RoboDK station: MoveBill_V2.rdk

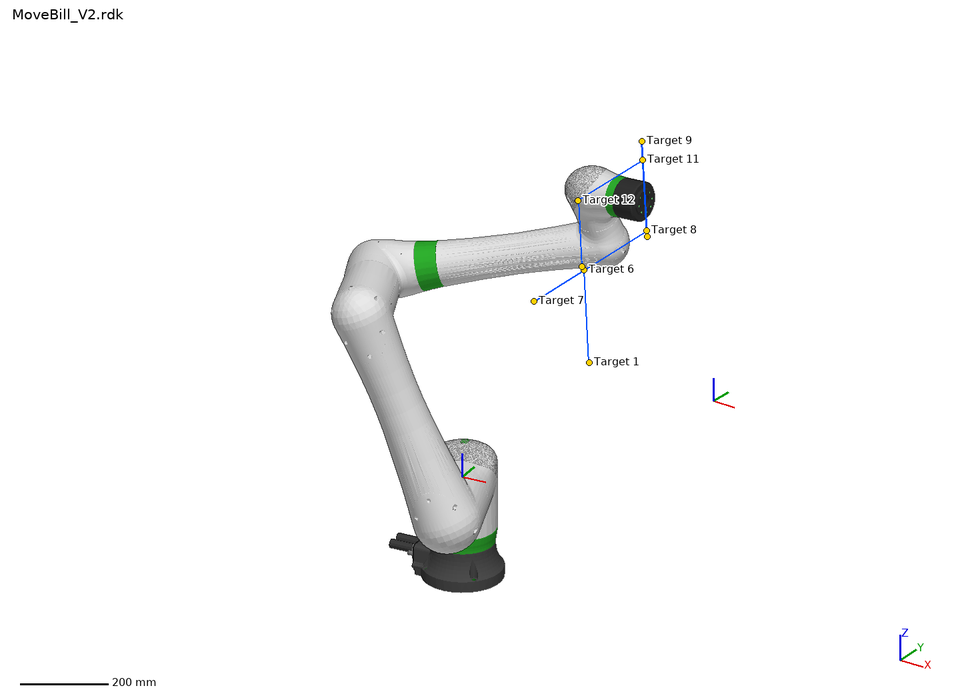
[picture v0: the station drawn from its stored meshes, robots at their saved joint values, targets as dots, program paths as lines]
Station MoveBill_V2 (saved by RoboDK 5.5.4). Poses are relative to the parent item; angles as X-Y-Z fixed-axis rotations.
Station parameters (name, value as stored): LIN64
  - frame Fanuc CRX-10iA Base at (0, 0, 245) mm, rotated rx 0 ry 0 rz 7.43 deg
    - robot Fanuc CRX-10iA: 6 axes, payload 10 kg, reach 1249 mm, repeatability 0.05 mm, weight 40 kg
        modified DH rows (alpha deg, a mm, theta deg, d mm): 0, 0, 0, 245; -90, 0, -90, 0; 0, 540, 0, 0; -90, 0, 0, 540; 90, 0, 0, -150; -90, 0, 0, 160
        base shift (0, 0, -245) mm
        joint limits [-180, -180, -360, -190, -180, -190] to [180, 180, 430, 190, 180, 190]; home [0, 0, 0, 0, 0, 0]; saved at [18.103, -21.494, 12.7, 77.531, -27.627, -73.192]
  - frame Frame 2 at (800, -150, 720) mm
    - target Target 1 (Cartesian target) at (-344.12, 0, 0.97) mm, rotated rx 0 ry -90 rz -180 deg; joints [-7.434, -26.873, -0.606, -0.001, 0.606, 0.001] of Fanuc CRX-10iA
    - target Target 2 (Cartesian target) at (-344.12, 0, 0.97) mm, rotated rx 0 ry -58.74 rz -180 deg; joints [-7.434, -22.969, -11.131, 0, 42.396, 0] of Fanuc CRX-10iA
    - target Target 3 (Cartesian target) at (-344.12, 0, 0.97) mm, rotated rx -180 ry -70.85 rz 0 deg; joints [-7.434, -25.639, 4.421, 0, -23.569, 0] of Fanuc CRX-10iA
    - target Target 4 (Cartesian target) at (-344.12, 0, 0.97) mm, rotated rx 0 ry -62.75 rz -180 deg; joints [-7.434, -23.884, -9.706, 0, 36.952, 0] of Fanuc CRX-10iA
    - target Target 5 (Cartesian target) at (-344.12, 0, 0.97) mm, rotated rx -180 ry -44.83 rz 0 deg; joints [-50.405, -20.254, -0.149, 145.831, 58.825, -127.185] of Fanuc CRX-10iA
    - target Target 6 (Cartesian target) at (-358.03, 0, 231.21) mm, rotated rx 0 ry -86.54 rz 180 deg; joints [-36.371, -22.317, 5.067, 92.024, 28.899, -94.221] of Fanuc CRX-10iA
    - target Target 7 (Cartesian target) at (-358.03, -197.91, 231.21) mm, rotated rx 0 ry -86.54 rz 180 deg; joints [-57.288, -9.378, 1.493, 86.735, 49.841, -89.036] of Fanuc CRX-10iA
    - target Target 8 (Cartesian target) at (-358.03, 247.35, 231.21) mm, rotated rx 0 ry -86.54 rz -180 deg; joints [14.432, -24.419, 5.997, 84.347, -21.935, -82.523] of Fanuc CRX-10iA
    - target Target 9 (Cartesian target) at (-371.45, 247.35, 453.3) mm, rotated rx 0 ry -86.54 rz -180 deg; joints [28.744, -12.647, 31.715, 57.716, -44.184, -46.094] of Fanuc CRX-10iA
    - target Target 10 (Cartesian target) at (-357.19, 247.35, 217.34) mm, rotated rx 0 ry -86.54 rz -180 deg; joints [12.79, -24.851, 4.601, 87.51, -20.205, -86.074] of Fanuc CRX-10iA
    - target Target 11 (Cartesian target) at (-368.66, 247.35, 407.03) mm, rotated rx 0 ry -86.54 rz -180 deg; joints [26.686, -16.069, 25.782, 61.412, -39.616, -52.383] of Fanuc CRX-10iA
    - target Target 12 (Cartesian target) at (-368.66, -8.23, 407.03) mm, rotated rx 0 ry -86.54 rz -180 deg; joints [-9.194, -14.506, 41.138, -2.873, -37.714, 2.168] of Fanuc CRX-10iA
    - target Target 13 (Cartesian target) at (-358.7, -8.23, 242.24) mm, rotated rx 0 ry -86.54 rz -180 deg; joints [-9.208, -23.009, 24.319, -4.962, -20.931, 4.529] of Fanuc CRX-10iA
  - Python program testCRX10Model_10 (listed below)
  - Python program Prog2 (listed below)
  - program Prog3 (14 instructions, listed below)
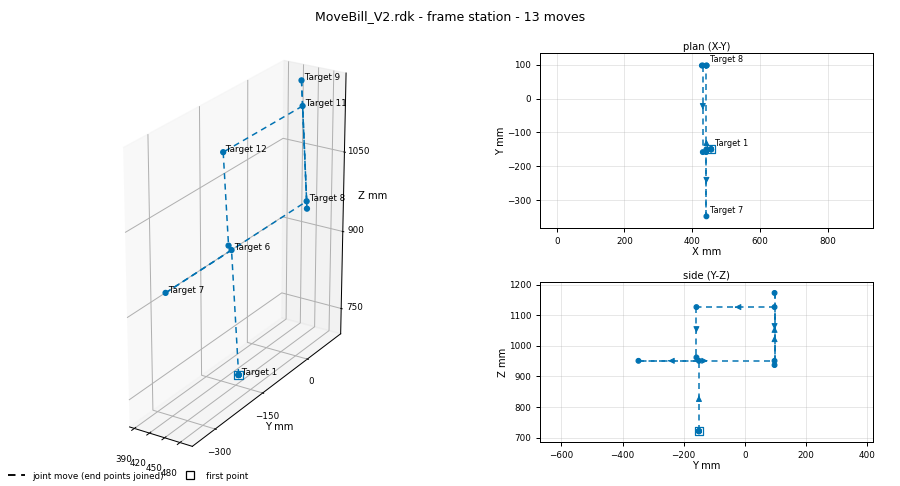
[picture p0: tool path of MoveBill_V2.rdk in frame station, 13 of 13 moves have a stored position in this frame; points joined in program order, loops and branches not executed]

--- Python program testCRX10Model_10 ---
import time

from robodk.robolink import *                  # import the robolink library
RDK = Robolink()                        # connect to the RoboDK API (RoboDK starts if it has not started

robots = RDK.ItemList(ITEM_TYPE_ROBOT)
print(robots)


# tool  = RDK.Item('SCHUNK- 1321170 Co-act EGP-C 40-N-N-KTOE_ 0')                # Get an item named Tool (name in the RoboDK station tree)

robot = RDK.Item('', ITEM_TYPE_ROBOT)   # Get the first available robot


robot.Connect()
RDK.setRunMode(RUNMODE_RUN_ROBOT)
#RDK.setRunMode(RUNMODE_SIMULATE)
#frame = RDK.ItemUserPick('Select a reference frame', ITEM_TYPE_FRAME)   # Promt the user to select a reference frame
frame = RDK.Item('Frame 2', ITEM_TYPE_FRAME)

robot.setPoseFrame(frame)
# robot.setPoseTool(tool)

robot.setSpeed(speed_joints = 1000, speed_linear = 1000, accel_linear = 1000, accel_joints = 1000)

for i in range(0,3):
	print("Run: ", i)
	target = RDK.Item('Back', ITEM_TYPE_TARGET)   # Get a target called "turn1"
	robot.MoveJ(target)             # Move the robot to the target using the selected reference frame

	#time.sleep(1.0)

	target = RDK.Item('Fwd', ITEM_TYPE_TARGET)   # Get a target called "home"
	robot.MoveJ(target)             # Move the robot to the target using the selected reference frame



	target = RDK.Item('Back', ITEM_TYPE_TARGET)   # Get a target called "home"
	robot.MoveJ(target)             # Move the robot to the target using the selected reference frame



	target = RDK.Item('Fwd', ITEM_TYPE_TARGET)   # Get a target called "home"
	robot.MoveJ(target)             # Move the robot to the target using the selected reference frame

#	target = RDK.Item('Home', ITEM_TYPE_TARGET)   # Get a target called "home"
#	robot.MoveJ(target)             # Move the robot to the target using the selected reference frame

--- Python program Prog2 ---
# Type help("robodk.robolink") or help("robodk.robomath") for more information
# Press F5 to run the script
# Documentation: https://robodk.com/doc/en/RoboDK-API.html
# Reference:     https://robodk.com/doc/en/PythonAPI/robodk.html
# Note: It is not required to keep a copy of this file, your Python script is saved with your RDK project

# You can also use the new version of the API:
from robodk import robolink    # RoboDK API
from robodk import robomath    # Robot toolbox
RDK = robolink.Robolink()

# Forward and backwards compatible use of the RoboDK API:
# Remove these 2 lines to follow python programming guidelines
from robodk import *      # RoboDK API
from robolink import *    # Robot toolbox
# Link to RoboDK
# RDK = Robolink()

# Notify user:
print('To edit this program:\nright click on the Python program, then, select "Edit Python script"')

# Program example:
item = RDK.Item('base')
if item.Valid():
    print('Item selected: ' + item.Name())
    print('Item posistion: ' + repr(item.Pose()))

print('Items in the station:')
itemlist = RDK.ItemList()
print(itemlist)

# Provoking an exception will display the console output if you run this script from RoboDK
raise Exception('Program not edited.')

--- program Prog3 (robot Fanuc CRX-10iA) ---
  Set Ref.: Frame 2
  MoveJ (Target 1)
  MoveJ (Target 2)
  MoveJ (Target 3)
  MoveJ (Target 4)
  MoveJ (Target 5)
  MoveJ (Target 6)
  MoveJ (Target 7)
  MoveJ (Target 8)
  MoveJ (Target 9)
  MoveJ (Target 10)
  MoveJ (Target 11)
  MoveJ (Target 12)
  MoveJ (Target 13)
